INTERFACE I_Drive_Type_1_Axis

METHOD Drive : BOOL
VAR_INPUT
END_VAR
END_METHOD

PROPERTY Position : real
GET
END_GET
SET
END_SET
END_PROPERTY

END_INTERFACE

(* stored: Version 1.1.0.1, ProductVersion 3.1.4024.15
   Itf I_Drive_Type_1_Axis: Id {b4fc8472-a3e3-4a62-8eaa-4b1914b96dc9}
   Method Drive: Id {77ce58b4-7975-422a-862d-7785438f932e}
   Property Position: Id {b3bd2303-8353-4695-8764-831b802e4171}
   Get Get: Id {1c2f0225-5620-4a11-87bf-b800f391da16}
   Set Set: Id {87d49c64-5f25-4f2d-84d1-0c084945ec06} *)
